(* PLC project DCMotor, Dassault Systèmes orchideo | easySSP (eXXcellent solutions GmbH) orchideo | easySSP (eXXcellent solutions GmbH) *)
(* stored: creationDateTime 2024-02-06T13:21:37Z, contentDescription SystemStructure.ssd *)

FUNCTION_BLOCK stimuli_model
  VAR_OUTPUT
    U : REAL := 0.0;
    M_load : REAL := 0.0;
  END_VAR


ACTION C_source_code:

END_ACTION
END_FUNCTION_BLOCK

FUNCTION_BLOCK edrive_mass
  VAR_INPUT
    M_A : REAL := 0.0;
    M_B : REAL := 0.0;
  END_VAR
  VAR_OUTPUT
    phiB : REAL := 0.0;
    wB : REAL := 0.0;
    wA : REAL := 0.0;
    phiA : REAL := 0.0;
  END_VAR


ACTION C_source_code:

END_ACTION
END_FUNCTION_BLOCK

FUNCTION_BLOCK emachine_model
  VAR_INPUT
    U : REAL := 0.0;
    w : REAL := 0.0;
    phi : REAL := 0.0;
  END_VAR
  VAR_OUTPUT
    M : REAL := 0.0;
    I : REAL := 0.0;
  END_VAR


ACTION C_source_code:

END_ACTION
END_FUNCTION_BLOCK

PROGRAM SuT
  VAR_INPUT
    M_load : REAL := 0.0;
    U : REAL := 0.0;
  END_VAR
  VAR_OUTPUT
    wB : REAL := 0.0;
    phiB : REAL := 0.0;
    M_mot : REAL := 0.0;
    I : REAL := 0.0;
  END_VAR

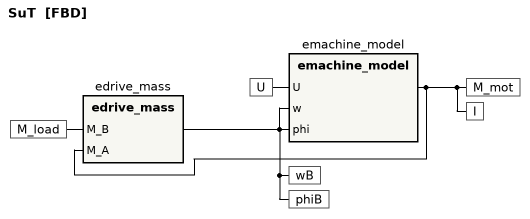
(* FBD diagram, written out as Structured Text *)
emachine_model(U := U, w := edrive_mass.wA, phi := edrive_mass.phiA);
edrive_mass(M_B := M_load, M_A := emachine_model.M);
wB := edrive_mass.wB;
phiB := edrive_mass.phiB;
M_mot := emachine_model.M;
I := emachine_model.I;
END_PROGRAM

PROGRAM DCMotor.DCMotor
  VAR_OUTPUT
    M_mot : REAL := 0.0;
    wB : REAL := 0.0;
    U : REAL := 0.0;
    I : REAL := 0.0;
  END_VAR

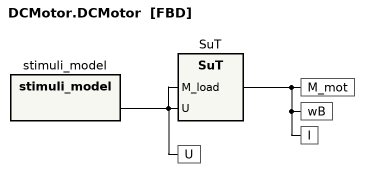
(* FBD diagram, written out as Structured Text *)
stimuli_model();
SuT(M_load := stimuli_model.M_load, U := stimuli_model.U);
M_mot := SuT.M_mot;
wB := SuT.wB;
U := stimuli_model.U;
I := SuT.I;
END_PROGRAM
